// TIA Portal V17 export
// export: Created 2023-03-06T08:28:50.7583733Z, ExportSetting WithDefaults, DisplayName Totally Integrated Automation Portal, DisplayVersion V17 Update 4, DisplayName TIA Portal Openness, DisplayVersion V17 Update 4, DisplayName TIA Portal Version Control Interface, DisplayVersion V17, DisplayName STEP 7 Professional, DisplayVersion V17 Update 4, DisplayName STEP 7 Safety, DisplayVersion V17, DisplayName WinCC Professional, DisplayVersion V17 Update 4
DATA_BLOCK "BMS2"   // DB21
{ S7_Optimized_Access := 'TRUE' }
VERSION : 0.1
// stored: AutoNumber false, DBAccessibleFromOPCUA true, DBAccessibleFromWebserver true, IsOnlyStoredInLoadMemory false, IsRetainMemResEnabled false, IsWriteProtectedInAS false, MemoryReserve 100
   VAR RETAIN
      TCON { S7_SetPoint := 'True'} : TCON_IP_v4;
   END_VAR
   VAR
      arrData : Array[1..125] of Word;
      xREQ : Bool;
      iCountDone : Int := 1;
      iCountRead : Int := 1;
      MBmode : USInt;
      MBdataAddr : UDInt;
      MBdataLen : UInt;
   END_VAR
   VAR RETAIN
      TCON10 { S7_SetPoint := 'True'} : TCON_IP_v4;
   END_VAR
   VAR
      arrData10 : Array[1..125] of Word;
      xREQ10 : Bool;
      iCountDone10 : Int := 1;
      iCountRead10 : Int := 1;
      MBmode10 : USInt;
      MBdataAddr10 : UDInt;
      MBdataLen10 : UInt;
   END_VAR
   VAR RETAIN
      TCON11 { S7_SetPoint := 'True'} : TCON_IP_v4;
   END_VAR
   VAR
      arrData11 : Array[1..125] of Word;
      xREQ11 : Bool;
      iCountDone11 : Int := 1;
      iCountRead11 : Int := 1;
      MBmode11 : USInt;
      MBdataAddr11 : UDInt;
      MBdataLen11 : UInt;
      BB { S7_SetPoint := 'True'} : "BMS_BB";
      BR01 { S7_SetPoint := 'True'} : "BMS_BR";
      BR02 { S7_SetPoint := 'True'} : "BMS_BR";
      BR03 { S7_SetPoint := 'True'} : "BMS_BR";
      BR04 { S7_SetPoint := 'True'} : "BMS_BR";
      BR05 { S7_SetPoint := 'True'} : "BMS_BR";
      BR06 { S7_SetPoint := 'True'} : "BMS_BR";
      BR07 { S7_SetPoint := 'True'} : "BMS_BR";
      BR08 { S7_SetPoint := 'True'} : "BMS_BR";
      BR09 { S7_SetPoint := 'True'} : "BMS_BR";
      BR10 { S7_SetPoint := 'True'} : "BMS_BR";
      BR11 { S7_SetPoint := 'True'} : "BMS_BR";
      BR12 { S7_SetPoint := 'True'} : "BMS_BR";
      TMS01 { S7_SetPoint := 'True'} : "BMS_TMS";
      TMS02 { S7_SetPoint := 'True'} : "BMS_TMS";
      TMS03 { S7_SetPoint := 'True'} : "BMS_TMS";
      TMS04 { S7_SetPoint := 'True'} : "BMS_TMS";
      TMS05 { S7_SetPoint := 'True'} : "BMS_TMS";
      TMS06 { S7_SetPoint := 'True'} : "BMS_TMS";
      TMS07 { S7_SetPoint := 'True'} : "BMS_TMS";
      TMS08 { S7_SetPoint := 'True'} : "BMS_TMS";
      TMS09 { S7_SetPoint := 'True'} : "BMS_TMS";
      TMS10 { S7_SetPoint := 'True'} : "BMS_TMS";
      TMS11 { S7_SetPoint := 'True'} : "BMS_TMS";
      TMS12 { S7_SetPoint := 'True'} : "BMS_TMS";
      rNomEnergyBank { S7_SetPoint := 'True'} : Real;
      rPbank : Real;
      rCrate : Real;
      rSOCavlCha : Real;
      rSOCavlDsch : Real;
      rEnergyAvlCha : Real;
      rEnergyAvlDsch : Real;
      diTimeEndCha : DInt;
      diTimeEndDsch : DInt;
      rVcellMinSet : Real := 2.76;
      rVcellMinReset : Real := 3.05;
      rVcellMaxSet : Real := 3.68;
      rVcellMaxReset : Real := 3.3;
      rVcellAutoChaSet : Real := 2.7;
      rVcellAutoChaReset : Real := 3.1;
      rPchaLim : Real;
      rPdschLim : Real;
      wRackFlt : Word;
      wRackOn : Word;
      xBankAvl : Bool;
      xEnbCha : Bool;
      xEnbDsch : Bool;
      xAutoChaCmd : Bool;
      xSwitchGearSt : Bool;
      xPwrOffReadySt : Bool;
      xPwrOnReadySt : Bool;
      xPwrOnFltSt : Bool;
      xPwrOffFltSt : Bool;
      xInitSt : Bool;
      xNormOpSt : Bool;
      xFullChaSt : Bool;
      xFullDschSt : Bool;
      xWarnSt : Bool;
      xFltSt : Bool;
      xInitCmd : Bool;
      xStayCmd : Bool;
      xCloseCmd : Bool;
      xOpenCmd : Bool;
      xFltClearCmd : Bool;
      wCmd : Word;
      wFltClearCmd : Word;
      BBwAlm1 : Word;
      BBwWarn1 : Word;
      BBxCommFltSt : Bool;
      BBxFltSt : Bool;
      BBxAlmSt : Bool;
      BBxWarnSt : Bool;
      BR01wAlm1 : Word;
      BR01wAlm2 : Word;
      BR01wAlm3 : Word;
      BR01wWarn1 : Word;
      BR01xFltSt : Bool;
      BR01xAlmSt : Bool;
      BR01xWarnSt : Bool;
      BR02wAlm1 : Word;
      BR02wAlm2 : Word;
      BR02wAlm3 : Word;
      BR02wWarn1 : Word;
      BR02xFltSt : Bool;
      BR02xAlmSt : Bool;
      BR02xWarnSt : Bool;
      BR03wAlm1 : Word;
      BR03wAlm2 : Word;
      BR03wAlm3 : Word;
      BR03wWarn1 : Word;
      BR03xFltSt : Bool;
      BR03xAlmSt : Bool;
      BR03xWarnSt : Bool;
      BR04wAlm1 : Word;
      BR04wAlm2 : Word;
      BR04wAlm3 : Word;
      BR04wWarn1 : Word;
      BR04xFltSt : Bool;
      BR04xAlmSt : Bool;
      BR04xWarnSt : Bool;
      BR05wAlm1 : Word;
      BR05wAlm2 : Word;
      BR05wAlm3 : Word;
      BR05wWarn1 : Word;
      BR05xFltSt : Bool;
      BR05xAlmSt : Bool;
      BR05xWarnSt : Bool;
      BR06wAlm1 : Word;
      BR06wAlm2 : Word;
      BR06wAlm3 : Word;
      BR06wWarn1 : Word;
      BR06xFltSt : Bool;
      BR06xAlmSt : Bool;
      BR06xWarnSt : Bool;
      BR07wAlm1 : Word;
      BR07wAlm2 : Word;
      BR07wAlm3 : Word;
      BR07wWarn1 : Word;
      BR07xFltSt : Bool;
      BR07xAlmSt : Bool;
      BR07xWarnSt : Bool;
      BR08wAlm1 : Word;
      BR08wAlm2 : Word;
      BR08wAlm3 : Word;
      BR08wWarn1 : Word;
      BR08xFltSt : Bool;
      BR08xAlmSt : Bool;
      BR08xWarnSt : Bool;
      BR09wAlm1 : Word;
      BR09wAlm2 : Word;
      BR09wAlm3 : Word;
      BR09wWarn1 : Word;
      BR09xFltSt : Bool;
      BR09xAlmSt : Bool;
      BR09xWarnSt : Bool;
      BR10wAlm1 : Word;
      BR10wAlm2 : Word;
      BR10wAlm3 : Word;
      BR10wWarn1 : Word;
      BR10xFltSt : Bool;
      BR10xAlmSt : Bool;
      BR10xWarnSt : Bool;
      BR11wAlm1 : Word;
      BR11wAlm2 : Word;
      BR11wAlm3 : Word;
      BR11wWarn1 : Word;
      BR11xFltSt : Bool;
      BR11xAlmSt : Bool;
      BR11xWarnSt : Bool;
      BR12wAlm1 : Word;
      BR12wAlm2 : Word;
      BR12wAlm3 : Word;
      BR12wWarn1 : Word;
      BR12xFltSt : Bool;
      BR12xAlmSt : Bool;
      BR12xWarnSt : Bool;
      iNRackFault : Int;
      BR01xSSFltSt : Bool;
      BR02xSSFltSt : Bool;
      BR03xSSFltSt : Bool;
      BR04xSSFltSt : Bool;
      BR05xSSFltSt : Bool;
      BR06xSSFltSt : Bool;
      BR07xSSFltSt : Bool;
      BR08xSSFltSt : Bool;
      BR09xSSFltSt : Bool;
      BR10xSSFltSt : Bool;
      BR11xSSFltSt : Bool;
      BR12xSSFltSt : Bool;
   END_VAR
BEGIN
   TCON.RemoteAddress.ADDR[1] := 192;
   TCON.RemoteAddress.ADDR[2] := 168;
   TCON.RemoteAddress.ADDR[3] := 150;
   TCON.RemoteAddress.ADDR[4] := 44;
   TCON10.RemoteAddress.ADDR[1] := 192;
   TCON10.RemoteAddress.ADDR[2] := 168;
   TCON10.RemoteAddress.ADDR[3] := 150;
   TCON10.RemoteAddress.ADDR[4] := 44;
   TCON11.RemoteAddress.ADDR[1] := 192;
   TCON11.RemoteAddress.ADDR[2] := 168;
   TCON11.RemoteAddress.ADDR[3] := 150;
   TCON11.RemoteAddress.ADDR[4] := 44;
   BB.iNBRtotalCount := 10;
END_DATA_BLOCK
